FUNCTION_BLOCK FutureMCPowerCreator IMPLEMENTS I_TaskCreator
VAR_INPUT
END_VAR
VAR_OUTPUT
END_VAR
VAR
	_axis: REFERENCE TO AXIS_REF;
	_override: LREAL := 100.0;
	_enable_positive:	BOOL := TRUE; 
	_enable_negative:	BOOL := TRUE;
	_option : ST_PowerOptions;
	_buffer_mode : MC_BufferMode;
	_status : BOOL;
END_VAR

METHOD create_future : I_Future
VAR_INPUT
	(* Specify future name*)
	future_name	: STRING;
END_VAR
VAR
	_p_future : POINTER TO FutureMCPower;
END_VAR
_p_future := __NEW(FutureMCPower);
_p_future^.future_name := future_name;
_p_future^.set_parameters(_axis, _status);
_p_future^.set_options(_enable_positive, _enable_negative, _override, _buffer_mode, _option);
create_future := _p_future^;
END_METHOD

METHOD destroy_future : I_Future
VAR_INPUT
	(* Specify future instance whtat you want to delete.*)
	future	: I_Future;
END_VAR
VAR
	_p_future : POINTER TO FutureMCPower;
END_VAR
IF __QUERYPOINTER(future, _p_future) THEN
	__DELETE(_p_future);
	IF _p_future = 0  THEN
		destroy_future := 0;
	END_IF
END_IF
END_METHOD

METHOD set_options : BOOL
VAR_INPUT
	Enable_Positive:	BOOL; 
	Enable_Negative:	BOOL;
	Override:			LREAL := 100;
	buffer_mode : MC_BufferMode;
	option : ST_PowerOptions;
END_VAR
_override := Override;
_enable_positive := Enable_Positive;
_enable_negative := Enable_Negative;
_buffer_mode := buffer_mode;
_option := option;
END_METHOD

METHOD set_parameters : BOOL
VAR_INPUT
	axis : REFERENCE TO AXIS_REF;
	status : BOOL;
END_VAR
_axis REF= axis;
_status := status;
END_METHOD

END_FUNCTION_BLOCK

(* stored: Version 1.1.0.1, ProductVersion 3.1.4026.17
   POU FutureMCPowerCreator: Id {e49d35f1-eac8-4a7a-ac81-58af9d64cecc}, SpecialFunc None
   Method create_future: Id {a300494e-4c4b-4b5a-b968-720d096df000}
   Method destroy_future: Id {9fd6631a-522f-4043-a177-993b0c9aa8fc}
   Method set_options: Id {c98fe1a0-d780-444c-a3d7-5a90b0bbc16b}
   Method set_parameters: Id {f89aafbd-4c5a-459e-b519-0fa9196fc7ba} *)
